SUBAPPLICATION AX_SoftkeyToggle_RS_TO_AX_BG_PUBLISH (* Wraps AX_SoftkeyToggle_RS_TO_AX (Toggle/Reset-Zustand: SoftKey ODER AUX ODER lokale Web-/Dashboard-Methode ODER IO-Diag-Testbutton fuer den Toggle, SoftKey ODER AUX ODER Methode fuer den Reset) und treibt daraus Hintergrundfarbe (SoftKey+AUX aus 1 GreenWhiteBackground3_AX) + lokalen State-Publish - OHNE physischen Ausgang (Gegenstueck zu AX_SoftkeyToggle_RS_TO_QXA_BG, das zusaetzlich noch 1 logiBUS_QXA treibt). Fuer Faelle, in denen der Toggle-Zustand vom Aufrufer noch weiterverarbeitet wird, bevor er auf einen oder mehrere physische Ausgaenge geht (z.B. Baender-Sequenzierung: Taste 5 toggelt, danach erst AX_TON/AX_TOF pro Kanal). Toggle-Zustand bleibt zusaetzlich als Plug OUT verfuegbar. *)
  (* Standard: 61499-2; Description: Copyright (c) 2026 Meisterschulen am Ostbahnhof This program and the accompanying materials are made available under the terms of the Eclipse Public License 2.0 which is available at https://www.eclipse.org/legal/epl-2.0/ SPDX-License-Identifier: EPL-2.0 *)
  (* Version 1.3, 2026-09-16, Franz Höpfinger, Meisterschulen am Ostbahnhof, Event-Input RESET in AUS umbenannt (Franz: 'der Eingang soll AUS heissen'), Durchreiche an ToggleState.AUS (AX_SoftkeyToggle_RS_TO_AX v1.4). *)
  (* Version 1.2, 2026-09-16, Franz Höpfinger, Meisterschulen am Ostbahnhof, Event-Input RESET durchgereicht an ToggleState.RESET (AX_SoftkeyToggle_RS_TO_AX v1.3) - rein additiv, fuer einen zentral gelesenen gemeinsamen SoftKey. *)
  (* Version 1.1, 2026-09-15, Franz Höpfinger, Meisterschulen am Ostbahnhof, FORCE_OFF Socket (AX) ergaenzt - reiner Durchreich-Socket an ToggleState.FORCE_OFF (AX_SoftkeyToggle_RS_TO_AX v1.2). Fuer eine uebergeordnete Sicherheitsabschaltung (z.B. Zapfwelle_Ueberwachung, KVE14 Zeile 33) - rein additiv, bestehende Instanzen muessen den neuen Socket verdrahten (z.B. auf einen festen FALSE-Literal, wenn nicht gebraucht). *)
  (* Version 1.0, 2026-09-15, Franz Höpfinger, Meisterschulen am Ostbahnhof, initial implementation - aus Baender_EinAus.SUB herausgeloest (ToggleState/AX_SPLIT_4-Anteil fuer Background+Publish/GreenWhiteBackground_AX/PUBLISH_STATE, Franz: 'GreenWhiteBackground3_AX AX_SoftkeyToggle_RS_TO_AX koennen zusammen in eine SUB, PUBLISH_STATE kann da auch rein'). TOF_IgelElevator/TON_Querband-Staffelung bleibt beim Aufrufer, da die 2 zeitversetzten Ausgaenge ausserhalb dieser SUB liegen. *)
  PACKAGE MyLib::sys;
  IMPORT isobus::UT::Q::const::IDs::ID_NULL;
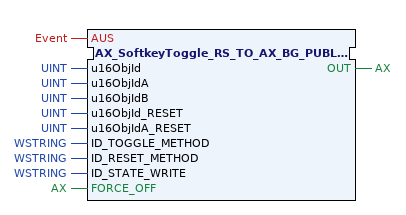
  EVENT_INPUT
    AUS; (* Reset hart auf AUS, von aussen als Event (z.B. 1 zentral gelesener gemeinsamer SoftKey) - Durchreiche an ToggleState.AUS. Unverdrahtet lassen, wenn nicht gebraucht. *)
  END_EVENT
  VAR_INPUT
    u16ObjId : UINT := ID_NULL; (* Object ID Softkey Ein/Aus (Toggle), traegt auch die Hintergrundfarbe *)
    u16ObjIdA : UINT := ID_NULL; (* Object ID AuxFunction2 (Joystick) fuer den Toggle - gleichberechtigt zum SoftKey, zeigt Hintergrundfarbe am Aux-Handle mit *)
    u16ObjIdB : UINT := ID_NULL; (* Object ID IO-Diag-Testbutton (Ausgaenge-Diagnoseseite) - toggelt gleichberechtigt mit (keine eigene Hintergrundfarbe, GreenWhiteBackground3_AX kennt nur SoftKey+AUX) *)
    u16ObjId_RESET : UINT := ID_NULL; (* Object ID Softkey 'Alles Aus' (Reset, hart auf AUS) - z.B. SoftKey_AUS *)
    u16ObjIdA_RESET : UINT := ID_NULL; (* Object ID AuxFunction2 (Joystick) fuer den Reset - gleichberechtigt zum Softkey 'Alles Aus' *)
    ID_TOGGLE_METHOD : WSTRING; (* Lokale Methodenadresse (ACTION=CREATE_METHOD) fuer den argumentlosen Toggle-Trigger - wird von Web-Client (vt-ui-mirror) UND direkt vom OPC-Dashboard aufgerufen *)
    ID_RESET_METHOD : WSTRING; (* Lokale Methodenadresse (ACTION=CREATE_METHOD) fuer den argumentlosen Reset-Trigger (hart auf AUS) - wird von Web-Client UND OPC-Dashboard aufgerufen *)
    ID_STATE_WRITE : WSTRING; (* Lokale Publish-Adresse (ACTION=WRITE) fuer den tatsaechlichen Toggle-Zustand (AX_T_FF_SR.Q) - wird von Web-Client/Dashboard remote abonniert *)
  END_VAR
  SOCKETS
    FORCE_OFF : adapter::types::unidirectional::AX; (* Optional: steigende Flanke resettet hart auf AUS (z.B. Sicherheitsabschaltung) - reiner Durchreich-Socket an ToggleState.FORCE_OFF. Unverdrahtet lassen (fester FALSE-Literal), wenn nicht gebraucht. *)
  END_SOCKETS
  PLUGS
    OUT : adapter::types::unidirectional::AX; (* Toggle-Zustand (AX_T_FF_SR.Q) - fuer Weiterverarbeitung beim Aufrufer (z.B. AX_TON/AX_TOF-Staffelung), Hintergrund+Publish sind hier bereits erledigt *)
  END_PLUGS
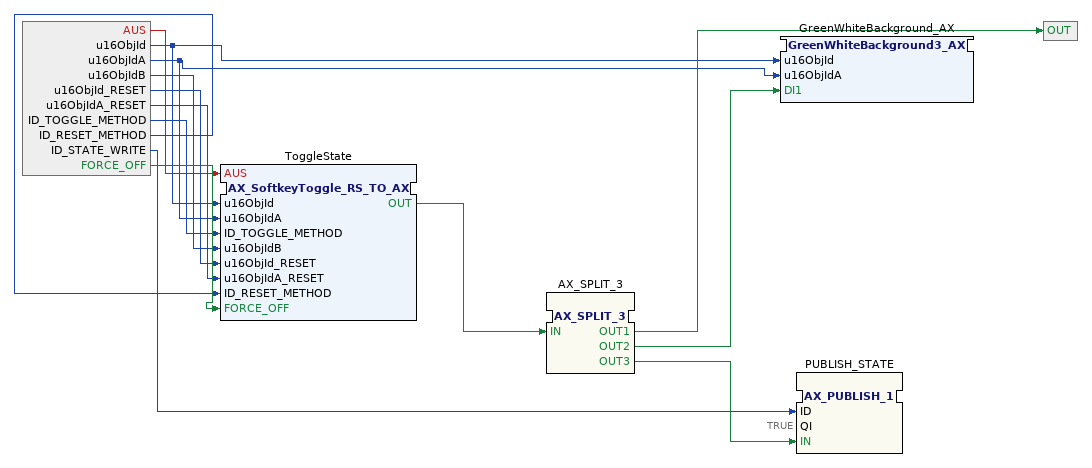
  FBS
    AX_SPLIT_3 : adapter::events::unidirectional::AX_SPLIT_3;
    PUBLISH_STATE : adapter::net::AX_PUBLISH_1(QI := TRUE);
  END_FBS
  SUBAPPS
    ToggleState : MyLib::sys::AX_SoftkeyToggle_RS_TO_AX;
    GreenWhiteBackground_AX : MyLib::sys::GreenWhiteBackground3_AX;
  END_SUBAPPS
  EVENT_CONNECTIONS
    AUS TO ToggleState.AUS;
  END_CONNECTIONS
  DATA_CONNECTIONS
    u16ObjId TO ToggleState.u16ObjId;
    u16ObjIdA TO ToggleState.u16ObjIdA;
    ID_TOGGLE_METHOD TO ToggleState.ID_TOGGLE_METHOD;
    u16ObjIdB TO ToggleState.u16ObjIdB;
    u16ObjId_RESET TO ToggleState.u16ObjId_RESET;
    u16ObjIdA_RESET TO ToggleState.u16ObjIdA_RESET;
    ID_RESET_METHOD TO ToggleState.ID_RESET_METHOD;
    u16ObjId TO GreenWhiteBackground_AX.u16ObjId;
    u16ObjIdA TO GreenWhiteBackground_AX.u16ObjIdA;
    ID_STATE_WRITE TO PUBLISH_STATE.ID;
  END_CONNECTIONS
  ADAPTER_CONNECTIONS
    ToggleState.OUT TO AX_SPLIT_3.IN;
    AX_SPLIT_3.OUT1 TO OUT;
    AX_SPLIT_3.OUT2 TO GreenWhiteBackground_AX.DI1;
    AX_SPLIT_3.OUT3 TO PUBLISH_STATE.IN;
    FORCE_OFF TO ToggleState.FORCE_OFF;
  END_CONNECTIONS
END_SUBAPPLICATION
